// TwinCAT 3 PLC project xpp_jjslit_motion
// ProgramVersion: 3.1.4022.7
// libraries:
//   lcls-twincat-motion, * (SLAC)
//   Tc2_Standard, * (Beckhoff Automation GmbH)
//   Tc2_System, * (Beckhoff Automation GmbH)
//   Tc3_Module, * (Beckhoff Automation GmbH)
// project tree:
//   / PlcTask.TcTTO (not stored)
//   POUs/ Main.TcPOU
// real-time tasks:
//   TASK PlcTask: cycle T#10ms, priority 20, ADS port 350
// motion (NC):
// I/O:
//   DEVICE Device 1 (EtherCAT), AmsNetId 172.21.84.130.1.1
//     JJ_PLC_EK1200
// variable links:
//   xpp_jjslit_motion Instance <-> Device 1 (EtherCAT)/JJ_PLC_EK1200/JJ_1_H_Gap_EL7037
//     PlcTask Inputs/Main.M3.bLimitBackwardEnable <-> STM Status/Status/Digital input 2
//     PlcTask Inputs/Main.M3.bLimitForwardEnable <-> STM Status/Status/Digital input 1
//   xpp_jjslit_motion Instance <-> Device 1 (EtherCAT)/JJ_PLC_EK1200/JJ_1_H_Offset_EL7031
//     PlcTask Inputs/Main.M4.bLimitBackwardEnable <-> STM Status/Status/Digital input 2
//     PlcTask Inputs/Main.M4.bLimitForwardEnable <-> STM Status/Status/Digital input 1
//   xpp_jjslit_motion Instance <-> Device 1 (EtherCAT)/JJ_PLC_EK1200/JJ_1_V_Gap_EL7037
//     PlcTask Inputs/Main.M1.bLimitBackwardEnable <-> STM Status/Status/Digital input 2
//     PlcTask Inputs/Main.M1.bLimitForwardEnable <-> STM Status/Status/Digital input 1
//   xpp_jjslit_motion Instance <-> Device 1 (EtherCAT)/JJ_PLC_EK1200/JJ_1_V_Offset_EL7037
//     PlcTask Inputs/Main.M2.bLimitBackwardEnable <-> STM Status/Status/Digital input 2
//     PlcTask Inputs/Main.M2.bLimitForwardEnable <-> STM Status/Status/Digital input 1
//   xpp_jjslit_motion Instance <-> Device 1 (EtherCAT)/JJ_PLC_EK1200/JJ_2_H_Gap_EL7037
//     PlcTask Inputs/Main.M7.bLimitBackwardEnable <-> STM Status/Status/Digital input 2
//     PlcTask Inputs/Main.M7.bLimitForwardEnable <-> STM Status/Status/Digital input 1
//   xpp_jjslit_motion Instance <-> Device 1 (EtherCAT)/JJ_PLC_EK1200/JJ_2_H_Offset_EL7037
//     PlcTask Inputs/Main.M8.bLimitBackwardEnable <-> STM Status/Status/Digital input 2
//     PlcTask Inputs/Main.M8.bLimitForwardEnable <-> STM Status/Status/Digital input 1
//   xpp_jjslit_motion Instance <-> Device 1 (EtherCAT)/JJ_PLC_EK1200/JJ_2_V_Gap_EL7037
//     PlcTask Inputs/Main.M5.bLimitBackwardEnable <-> STM Status/Status/Digital input 2
//     PlcTask Inputs/Main.M5.bLimitForwardEnable <-> STM Status/Status/Digital input 1
//   xpp_jjslit_motion Instance <-> Device 1 (EtherCAT)/JJ_PLC_EK1200/JJ_2_V_Offset_EL7037
//     PlcTask Inputs/Main.M6.bLimitBackwardEnable <-> STM Status/Status/Digital input 2
//     PlcTask Inputs/Main.M6.bLimitForwardEnable <-> STM Status/Status/Digital input 1
//   xpp_jjslit_motion Instance <-> Device 1 (EtherCAT)/JJ_PLC_EK1200/JJ_3_H_Gap_EL7037
//     PlcTask Inputs/Main.M11.bLimitBackwardEnable <-> STM Status/Status/Digital input 2
//     PlcTask Inputs/Main.M11.bLimitForwardEnable <-> STM Status/Status/Digital input 1
//   xpp_jjslit_motion Instance <-> Device 1 (EtherCAT)/JJ_PLC_EK1200/JJ_3_H_Offset_EL7037
//     PlcTask Inputs/Main.M12.bLimitBackwardEnable <-> STM Status/Status/Digital input 2
//     PlcTask Inputs/Main.M12.bLimitForwardEnable <-> STM Status/Status/Digital input 1
//   xpp_jjslit_motion Instance <-> Device 1 (EtherCAT)/JJ_PLC_EK1200/JJ_3_V_Gap_EL7037
//     PlcTask Inputs/Main.M9.bLimitBackwardEnable <-> STM Status/Status/Digital input 2
//     PlcTask Inputs/Main.M9.bLimitForwardEnable <-> STM Status/Status/Digital input 1
//   xpp_jjslit_motion Instance <-> Device 1 (EtherCAT)/JJ_PLC_EK1200/JJ_3_V_Offset_EL7037
//     PlcTask Inputs/Main.M10.bLimitBackwardEnable <-> STM Status/Status/Digital input 2
//     PlcTask Inputs/Main.M10.bLimitForwardEnable <-> STM Status/Status/Digital input 1
//   xpp_jjslit_motion Instance <-> Device 1 (EtherCAT)/JJ_PLC_EK1200/JJ_4_H_Gap_EL7037
//     PlcTask Inputs/Main.M15.bLimitBackwardEnable <-> STM Status/Status/Digital input 2
//     PlcTask Inputs/Main.M15.bLimitForwardEnable <-> STM Status/Status/Digital input 1
//   xpp_jjslit_motion Instance <-> Device 1 (EtherCAT)/JJ_PLC_EK1200/JJ_4_H_Offset_EL7037
//     PlcTask Inputs/Main.M16.bLimitBackwardEnable <-> STM Status/Status/Digital input 2
//     PlcTask Inputs/Main.M16.bLimitForwardEnable <-> STM Status/Status/Digital input 1
//   xpp_jjslit_motion Instance <-> Device 1 (EtherCAT)/JJ_PLC_EK1200/JJ_4_V_Gap_EL7037
//     PlcTask Inputs/Main.M13.bLimitBackwardEnable <-> STM Status/Status/Digital input 2
//     PlcTask Inputs/Main.M13.bLimitForwardEnable <-> STM Status/Status/Digital input 1
//   xpp_jjslit_motion Instance <-> Device 1 (EtherCAT)/JJ_PLC_EK1200/JJ_4_V_Offset_EL7037
//     PlcTask Inputs/Main.M14.bLimitBackwardEnable <-> STM Status/Status/Digital input 2
//     PlcTask Inputs/Main.M14.bLimitForwardEnable <-> STM Status/Status/Digital input 1
//   xpp_jjslit_motion Instance <-> NC-Task 1 SAF/Axes/JJ_1_H_Gap
//     PlcTask Inputs/Main.M3.Axis.NcToPlc <-> Outputs/ToPlc
//     PlcTask Outputs/Main.M3.Axis.PlcToNc <-> Inputs/FromPlc
//   xpp_jjslit_motion Instance <-> NC-Task 1 SAF/Axes/JJ_1_H_Offset
//     PlcTask Inputs/Main.M4.Axis.NcToPlc <-> Outputs/ToPlc
//     PlcTask Outputs/Main.M4.Axis.PlcToNc <-> Inputs/FromPlc
//   xpp_jjslit_motion Instance <-> NC-Task 1 SAF/Axes/JJ_1_V_Gap
//     PlcTask Inputs/Main.M1.Axis.NcToPlc <-> Outputs/ToPlc
//     PlcTask Outputs/Main.M1.Axis.PlcToNc <-> Inputs/FromPlc
//   xpp_jjslit_motion Instance <-> NC-Task 1 SAF/Axes/JJ_1_V_Offset
//     PlcTask Inputs/Main.M2.Axis.NcToPlc <-> Outputs/ToPlc
//     PlcTask Outputs/Main.M2.Axis.PlcToNc <-> Inputs/FromPlc
//   xpp_jjslit_motion Instance <-> NC-Task 1 SAF/Axes/JJ_2_H_Gap
//     PlcTask Inputs/Main.M7.Axis.NcToPlc <-> Outputs/ToPlc
//     PlcTask Outputs/Main.M7.Axis.PlcToNc <-> Inputs/FromPlc
//   xpp_jjslit_motion Instance <-> NC-Task 1 SAF/Axes/JJ_2_H_Offset
//     PlcTask Inputs/Main.M8.Axis.NcToPlc <-> Outputs/ToPlc
//     PlcTask Outputs/Main.M8.Axis.PlcToNc <-> Inputs/FromPlc
//   xpp_jjslit_motion Instance <-> NC-Task 1 SAF/Axes/JJ_2_V_Gap
//     PlcTask Inputs/Main.M5.Axis.NcToPlc <-> Outputs/ToPlc
//     PlcTask Outputs/Main.M5.Axis.PlcToNc <-> Inputs/FromPlc
//   xpp_jjslit_motion Instance <-> NC-Task 1 SAF/Axes/JJ_2_V_Offset
//     PlcTask Inputs/Main.M6.Axis.NcToPlc <-> Outputs/ToPlc
//     PlcTask Outputs/Main.M6.Axis.PlcToNc <-> Inputs/FromPlc
//   xpp_jjslit_motion Instance <-> NC-Task 1 SAF/Axes/JJ_3_H_Gap
//     PlcTask Inputs/Main.M11.Axis.NcToPlc <-> Outputs/ToPlc
//     PlcTask Outputs/Main.M11.Axis.PlcToNc <-> Inputs/FromPlc
//   xpp_jjslit_motion Instance <-> NC-Task 1 SAF/Axes/JJ_3_H_Offset
//     PlcTask Inputs/Main.M12.Axis.NcToPlc <-> Outputs/ToPlc
//     PlcTask Outputs/Main.M12.Axis.PlcToNc <-> Inputs/FromPlc
//   xpp_jjslit_motion Instance <-> NC-Task 1 SAF/Axes/JJ_3_V_Gap
//     PlcTask Inputs/Main.M9.Axis.NcToPlc <-> Outputs/ToPlc
//     PlcTask Outputs/Main.M9.Axis.PlcToNc <-> Inputs/FromPlc
//   xpp_jjslit_motion Instance <-> NC-Task 1 SAF/Axes/JJ_3_V_Offset
//     PlcTask Inputs/Main.M10.Axis.NcToPlc <-> Outputs/ToPlc
//     PlcTask Outputs/Main.M10.Axis.PlcToNc <-> Inputs/FromPlc
//   xpp_jjslit_motion Instance <-> NC-Task 1 SAF/Axes/JJ_4_H_Gap
//     PlcTask Inputs/Main.M15.Axis.NcToPlc <-> Outputs/ToPlc
//     PlcTask Outputs/Main.M15.Axis.PlcToNc <-> Inputs/FromPlc
//   xpp_jjslit_motion Instance <-> NC-Task 1 SAF/Axes/JJ_4_H_Offset
//     PlcTask Inputs/Main.M16.Axis.NcToPlc <-> Outputs/ToPlc
//     PlcTask Outputs/Main.M16.Axis.PlcToNc <-> Inputs/FromPlc
//   xpp_jjslit_motion Instance <-> NC-Task 1 SAF/Axes/JJ_4_V_Gap
//     PlcTask Inputs/Main.M13.Axis.NcToPlc <-> Outputs/ToPlc
//     PlcTask Outputs/Main.M13.Axis.PlcToNc <-> Inputs/FromPlc
//   xpp_jjslit_motion Instance <-> NC-Task 1 SAF/Axes/JJ_4_V_Offset
//     PlcTask Inputs/Main.M14.Axis.NcToPlc <-> Outputs/ToPlc
//     PlcTask Outputs/Main.M14.Axis.PlcToNc <-> Inputs/FromPlc

// ---- POUs/Main.TcPOU
PROGRAM Main
VAR
	// Motors
	{attribute 'TcLinkTo' := '.bLimitForwardEnable	:=TIIB[JJ_1_V_Gap_EL7037]^STM Status^Status^Digital input 1;
                              .bLimitBackwardEnable	:=TIIB[JJ_1_V_Gap_EL7037]^STM Status^Status^Digital input 2'}
	{attribute 'pytmc' := '
		pv: XPP:USR:JJ1:YWIDTH
	'}
	M1 : DUT_MotionStage := (bPowerSelf:=True,
//    nEnableMode:=ENUM_StageEnableMode.ALWAYS,
    nEnableMode:=ENUM_StageEnableMode.DURING_MOTION,
	nBrakeMode:= ENUM_StageBrakeMode.NO_BRAKE,
	nHomingMode := ENUM_EpicsHomeCmd.LOW_LIMIT); // JJ_1_Vertical_Gap

	fbMotionStageM1 : FB_MotionStage;
	

	
	{attribute 'TcLinkTo' := '.bLimitForwardEnable	:=TIIB[JJ_1_V_Offset_EL7037]^STM Status^Status^Digital input 1;
                              .bLimitBackwardEnable	:=TIIB[JJ_1_V_Offset_EL7037]^STM Status^Status^Digital input 2'}
	{attribute 'pytmc' := '
		pv: XPP:USR:JJ1:YCENTER
	'}
	M2 : DUT_MotionStage := (bPowerSelf:=True,
//	nEnableMode:=ENUM_StageEnableMode.ALWAYS,
    nEnableMode:=ENUM_StageEnableMode.DURING_MOTION,
	nBrakeMode:= ENUM_StageBrakeMode.NO_BRAKE,
    nHomingMode := ENUM_EpicsHomeCmd.LOW_LIMIT); // JJ_1_Vertical_Offset

	fbMotionStageM2 : FB_MotionStage;
	
	{attribute 'TcLinkTo' := '.bLimitForwardEnable	:=TIIB[JJ_1_H_Gap_EL7037]^STM Status^Status^Digital input 1;
                              .bLimitBackwardEnable	:=TIIB[JJ_1_H_Gap_EL7037]^STM Status^Status^Digital input 2'}
	{attribute 'pytmc' := '
		pv: XPP:USR:JJ1:XWIDTH
	'}
	M3 : DUT_MotionStage := (bPowerSelf:=True,
//	nEnableMode:=ENUM_StageEnableMode.ALWAYS,
    nEnableMode:=ENUM_StageEnableMode.DURING_MOTION,
	nBrakeMode:= ENUM_StageBrakeMode.NO_BRAKE,
	nHomingMode := ENUM_EpicsHomeCmd.LOW_LIMIT); // JJ_1_Horizontal_Gap

	fbMotionStageM3 : FB_MotionStage;
	
	{attribute 'TcLinkTo' := '.bLimitForwardEnable	:=TIIB[JJ_1_H_Offset_EL7031]^STM Status^Status^Digital input 1;
                              .bLimitBackwardEnable	:=TIIB[JJ_1_H_Offset_EL7031]^STM Status^Status^Digital input 2'}
	{attribute 'pytmc' := '
		pv: XPP:USR:JJ1:XCENTER
	'}
	M4 : DUT_MotionStage := (bPowerSelf:=True,
//	nEnableMode:=ENUM_StageEnableMode.ALWAYS,
    nEnableMode:=ENUM_StageEnableMode.DURING_MOTION,
	nBrakeMode:= ENUM_StageBrakeMode.NO_BRAKE,
	nHomingMode := ENUM_EpicsHomeCmd.LOW_LIMIT); // JJ_1_Horizontal_Offset

	fbMotionStageM4 : FB_MotionStage;
	
	{attribute 'TcLinkTo' := '.bLimitForwardEnable	:=TIIB[JJ_2_V_Gap_EL7037]^STM Status^Status^Digital input 1;
                              .bLimitBackwardEnable	:=TIIB[JJ_2_V_Gap_EL7037]^STM Status^Status^Digital input 2'}
	{attribute 'pytmc' := '
		pv: XPP:USR:JJ2:YWIDTH
	'}
	M5 : DUT_MotionStage := (bPowerSelf:=True,
// 	nEnableMode:=ENUM_StageEnableMode.ALWAYS,
    nEnableMode:=ENUM_StageEnableMode.DURING_MOTION,
	nBrakeMode:= ENUM_StageBrakeMode.NO_BRAKE,
	nHomingMode := ENUM_EpicsHomeCmd.LOW_LIMIT); // JJ_2_Vertical_Gap

	fbMotionStageM5 : FB_MotionStage;
	
	{attribute 'TcLinkTo' := '.bLimitForwardEnable	:=TIIB[JJ_2_V_Offset_EL7037]^STM Status^Status^Digital input 1;
                              .bLimitBackwardEnable	:=TIIB[JJ_2_V_Offset_EL7037]^STM Status^Status^Digital input 2'}
	{attribute 'pytmc' := '
		pv: XPP:USR:JJ2:YCENTER
	'}
	M6 : DUT_MotionStage := (bPowerSelf:=True,
//	nEnableMode:=ENUM_StageEnableMode.ALWAYS,
    nEnableMode:=ENUM_StageEnableMode.DURING_MOTION,
	nBrakeMode:= ENUM_StageBrakeMode.NO_BRAKE,
	nHomingMode := ENUM_EpicsHomeCmd.LOW_LIMIT); // JJ_2_Vertical_Offset
	fbMotionStageM6 : FB_MotionStage;
	
	{attribute 'TcLinkTo' := '.bLimitForwardEnable	:=TIIB[JJ_2_H_Gap_EL7037]^STM Status^Status^Digital input 1;
                              .bLimitBackwardEnable	:=TIIB[JJ_2_H_Gap_EL7037]^STM Status^Status^Digital input 2'}
	{attribute 'pytmc' := '
		pv: XPP:USR:JJ2:XWIDTH
	'}
	M7 : DUT_MotionStage := (bPowerSelf:=True,
//	nEnableMode:=ENUM_StageEnableMode.ALWAYS,
    nEnableMode:=ENUM_StageEnableMode.DURING_MOTION,
	nBrakeMode:= ENUM_StageBrakeMode.NO_BRAKE,
	nHomingMode := ENUM_EpicsHomeCmd.LOW_LIMIT); // JJ_2_Horizontal_Gap

	fbMotionStageM7 : FB_MotionStage;
	
	{attribute 'TcLinkTo' := '.bLimitForwardEnable	:=TIIB[JJ_2_H_Offset_EL7037]^STM Status^Status^Digital input 1;
                              .bLimitBackwardEnable	:=TIIB[JJ_2_H_Offset_EL7037]^STM Status^Status^Digital input 2'}
	{attribute 'pytmc' := '
		pv: XPP:USR:JJ2:XCENTER
	'}
	M8 : DUT_MotionStage := (bPowerSelf:=True,
//	nEnableMode:=ENUM_StageEnableMode.ALWAYS,
    nEnableMode:=ENUM_StageEnableMode.DURING_MOTION,
	nBrakeMode:= ENUM_StageBrakeMode.NO_BRAKE,
	nHomingMode := ENUM_EpicsHomeCmd.LOW_LIMIT); // JJ_2_Horizontal_Offset

	fbMotionStageM8 : FB_MotionStage;
	
	{attribute 'TcLinkTo' := '.bLimitForwardEnable	:=TIIB[JJ_3_V_Gap_EL7037]^STM Status^Status^Digital input 1;
                              .bLimitBackwardEnable	:=TIIB[JJ_3_V_Gap_EL7037]^STM Status^Status^Digital input 2'}
	{attribute 'pytmc' := '
		pv: XPP:USR:JJ3:YWIDTH
	'}
	M9 : DUT_MotionStage := (bPowerSelf:=True,
//	nEnableMode:=ENUM_StageEnableMode.ALWAYS,
    nEnableMode:=ENUM_StageEnableMode.DURING_MOTION,
	nBrakeMode:= ENUM_StageBrakeMode.NO_BRAKE,
	nHomingMode := ENUM_EpicsHomeCmd.LOW_LIMIT); // JJ_3_Vertical_Gap

	fbMotionStageM9 : FB_MotionStage;
	
	{attribute 'TcLinkTo' := '.bLimitForwardEnable	:=TIIB[JJ_3_V_Offset_EL7037]^STM Status^Status^Digital input 1;
                              .bLimitBackwardEnable	:=TIIB[JJ_3_V_Offset_EL7037]^STM Status^Status^Digital input 2'}
	{attribute 'pytmc' := '
		pv: XPP:USR:JJ3:YCENTER
	'}
	M10 : DUT_MotionStage := (bPowerSelf:=True,
//	nEnableMode:=ENUM_StageEnableMode.ALWAYS,
    nEnableMode:=ENUM_StageEnableMode.DURING_MOTION,
	nBrakeMode:= ENUM_StageBrakeMode.NO_BRAKE,
	nHomingMode := ENUM_EpicsHomeCmd.LOW_LIMIT); // JJ_3_Vertical_Offset

	fbMotionStageM10 : FB_MotionStage;
	
	{attribute 'TcLinkTo' := '.bLimitForwardEnable	:=TIIB[JJ_3_H_Gap_EL7037]^STM Status^Status^Digital input 1;
                              .bLimitBackwardEnable	:=TIIB[JJ_3_H_Gap_EL7037]^STM Status^Status^Digital input 2'}
	{attribute 'pytmc' := '
		pv: XPP:USR:JJ3:XWIDTH
	'}
	M11 : DUT_MotionStage := (bPowerSelf:=True,
//	nEnableMode:=ENUM_StageEnableMode.ALWAYS,
    nEnableMode:=ENUM_StageEnableMode.DURING_MOTION,
	nBrakeMode:= ENUM_StageBrakeMode.NO_BRAKE,
	nHomingMode := ENUM_EpicsHomeCmd.LOW_LIMIT); // JJ_3_Horizontal_Gap

	fbMotionStageM11 : FB_MotionStage;
	
	{attribute 'TcLinkTo' := '.bLimitForwardEnable	:=TIIB[JJ_3_H_Offset_EL7037]^STM Status^Status^Digital input 1;
                              .bLimitBackwardEnable	:=TIIB[JJ_3_H_Offset_EL7037]^STM Status^Status^Digital input 2'}
	{attribute 'pytmc' := '
		pv: XPP:USR:JJ3:XCENTER
	'}
	M12 : DUT_MotionStage := (bPowerSelf:=True,
//	nEnableMode:=ENUM_StageEnableMode.ALWAYS,
    nEnableMode:=ENUM_StageEnableMode.DURING_MOTION,
	nBrakeMode:= ENUM_StageBrakeMode.NO_BRAKE,
	nHomingMode := ENUM_EpicsHomeCmd.LOW_LIMIT); // JJ_3_Horizontal_Offset

	fbMotionStageM12 : FB_MotionStage;
	
	{attribute 'TcLinkTo' := '.bLimitForwardEnable	:=TIIB[JJ_4_V_Gap_EL7037]^STM Status^Status^Digital input 1;
                              .bLimitBackwardEnable	:=TIIB[JJ_4_V_Gap_EL7037]^STM Status^Status^Digital input 2'}
	{attribute 'pytmc' := '
		pv: XPP:USR:JJ4:YWIDTH
	'}
	M13 : DUT_MotionStage := (bPowerSelf:=True,
//	nEnableMode:=ENUM_StageEnableMode.ALWAYS,
    nEnableMode:=ENUM_StageEnableMode.DURING_MOTION,
	nBrakeMode:= ENUM_StageBrakeMode.NO_BRAKE,
	nHomingMode := ENUM_EpicsHomeCmd.LOW_LIMIT); // JJ_4_Vertical_Gap

	fbMotionStageM13 : FB_MotionStage;
	
	{attribute 'TcLinkTo' := '.bLimitForwardEnable	:=TIIB[JJ_4_V_Offset_EL7037]^STM Status^Status^Digital input 1;
                              .bLimitBackwardEnable	:=TIIB[JJ_4_V_Offset_EL7037]^STM Status^Status^Digital input 2'}
	{attribute 'pytmc' := '
		pv: XPP:USR:JJ4:YCENTER
	'}
	M14 : DUT_MotionStage := (bPowerSelf:=True,
//	nEnableMode:=ENUM_StageEnableMode.ALWAYS,
    nEnableMode:=ENUM_StageEnableMode.DURING_MOTION,
	nBrakeMode:= ENUM_StageBrakeMode.NO_BRAKE,
	nHomingMode := ENUM_EpicsHomeCmd.LOW_LIMIT); // JJ_4_Vertical_Offset

	fbMotionStageM14 : FB_MotionStage;
	
	{attribute 'TcLinkTo' := '.bLimitForwardEnable	:=TIIB[JJ_4_H_Gap_EL7037]^STM Status^Status^Digital input 1;
                              .bLimitBackwardEnable	:=TIIB[JJ_4_H_Gap_EL7037]^STM Status^Status^Digital input 2'}
	{attribute 'pytmc' := '
		pv: XPP:USR:JJ4:XWIDTH
	'}
	M15 : DUT_MotionStage := (bPowerSelf:=True,
//	nEnableMode:=ENUM_StageEnableMode.ALWAYS,
    nEnableMode:=ENUM_StageEnableMode.DURING_MOTION,
	nBrakeMode:= ENUM_StageBrakeMode.NO_BRAKE,
	nHomingMode := ENUM_EpicsHomeCmd.LOW_LIMIT); // JJ_4_Horizontal_Gap

	fbMotionStageM15 : FB_MotionStage;
	
	{attribute 'TcLinkTo' := '.bLimitForwardEnable	:=TIIB[JJ_4_H_Offset_EL7037]^STM Status^Status^Digital input 1;
                              .bLimitBackwardEnable	:=TIIB[JJ_4_H_Offset_EL7037]^STM Status^Status^Digital input 2'}
	{attribute 'pytmc' := '
		pv: XPP:USR:JJ4:XCENTER
	'}
	M16 : DUT_MotionStage := (bPowerSelf:=True,
//	nEnableMode:=ENUM_StageEnableMode.ALWAYS,
    nEnableMode:=ENUM_StageEnableMode.DURING_MOTION,
	nBrakeMode:= ENUM_StageBrakeMode.NO_BRAKE,
	nHomingMode := ENUM_EpicsHomeCmd.LOW_LIMIT); // JJ_4_Horizontal_Offset

	fbMotionStageM16 : FB_MotionStage;
END_VAR

// Hardware Enable
M1.bHardwareEnable := TRUE;
fbMotionStageM1(stMotionStage:=M1);

M2.bHardwareEnable := TRUE;
fbMotionStageM2(stMotionStage:=M2);

M3.bHardwareEnable := TRUE;
fbMotionStageM3(stMotionStage:=M3);

M4.bHardwareEnable := TRUE;
fbMotionStageM4(stMotionStage:=M4);

M5.bHardwareEnable := TRUE;
fbMotionStageM5(stMotionStage:=M5);

M6.bHardwareEnable := TRUE;
fbMotionStageM6(stMotionStage:=M6);

M7.bHardwareEnable := TRUE;
fbMotionStageM7(stMotionStage:=M7);

M8.bHardwareEnable := TRUE;
fbMotionStageM8(stMotionStage:=M8);

M9.bHardwareEnable := TRUE;
fbMotionStageM9(stMotionStage:=M9);

M10.bHardwareEnable := TRUE;
fbMotionStageM10(stMotionStage:=M10);

M11.bHardwareEnable := TRUE;
fbMotionStageM11(stMotionStage:=M11);

M12.bHardwareEnable := TRUE;
fbMotionStageM12(stMotionStage:=M12);

M13.bHardwareEnable := TRUE;
fbMotionStageM13(stMotionStage:=M13);

M14.bHardwareEnable := TRUE;
fbMotionStageM14(stMotionStage:=M14);

M15.bHardwareEnable := TRUE;
fbMotionStageM15(stMotionStage:=M15);

M16.bHardwareEnable := TRUE;
fbMotionStageM16(stMotionStage:=M16);

END_PROGRAM
